(* PLC project Unnamed, Unknown Unnamed 1 *)
(* stored: creationDateTime 2025-06-11T12:12:01, modificationDateTime 2025-06-11T12:47:44 *)

PROGRAM part2
  VAR
    PosX_b0 AT %IX0.0 : BOOL;
    PosX_b1 AT %IX0.1 : BOOL;
    PosX_b2 AT %IX0.2 : BOOL;
    PosX_b3 AT %IX0.3 : BOOL;
    PosY_b0 AT %IX0.4 : BOOL;
    PosY_b1 AT %IX0.5 : BOOL;
    PosY_b2 AT %IX0.6 : BOOL;
    PosY_b3 AT %IX0.7 : BOOL;
    TargetX_b0 AT %IX1.0 : BOOL;
    TargetX_b1 AT %IX1.1 : BOOL;
    TargetX_b2 AT %IX1.2 : BOOL;
    TargetX_b3 AT %IX1.3 : BOOL;
    TargetY_b0 AT %IX1.4 : BOOL;
    TargetY_b1 AT %IX1.5 : BOOL;
    TargetY_b2 AT %IX1.6 : BOOL;
    TargetY_b3 AT %IX1.7 : BOOL;
    MoveUp AT %QX0.0 : BOOL;
    MoveDown AT %QX0.1 : BOOL;
    MoveLeft AT %QX0.2 : BOOL;
    MoveRight AT %QX0.3 : BOOL;
  END_VAR
  VAR
    PosX_UINT : UINT;
    PosY_UINT : UINT;
  END_VAR

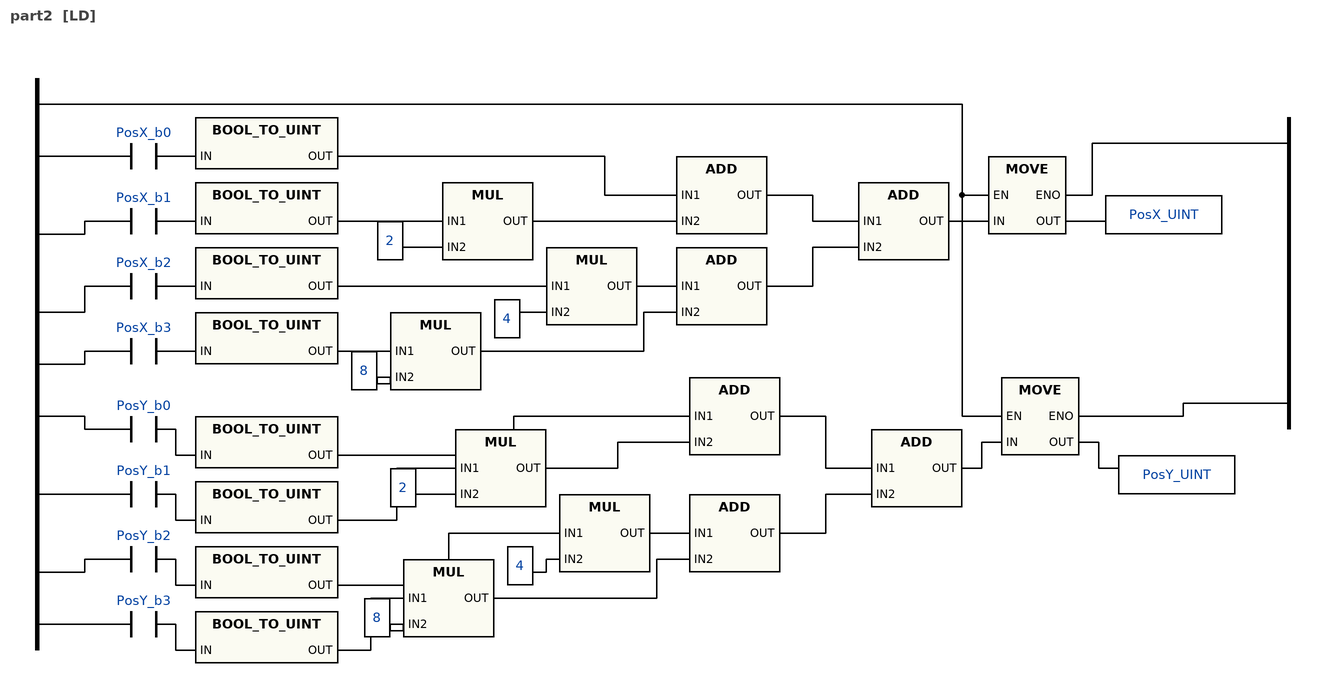
(* LD diagram, written out as Structured Text *)
PosX_UINT := BOOL_TO_UINT(PosX_b0) + BOOL_TO_UINT(PosX_b1) * 2 + (BOOL_TO_UINT(PosX_b2) * 4 + BOOL_TO_UINT(PosX_b3) * 8);
PosY_UINT := BOOL_TO_UINT(PosY_b0) + BOOL_TO_UINT(PosY_b1) * 2 + (BOOL_TO_UINT(PosY_b2) * 4 + BOOL_TO_UINT(PosY_b3) * 8);
END_PROGRAM

CONFIGURATION Config0
  RESOURCE Res0 ON PLC
    TASK task0(INTERVAL := T#20ms, PRIORITY := 0);
    PROGRAM instance0 WITH task0 : part2;
  END_RESOURCE
END_CONFIGURATION
